// TwinCAT 3 PLC project Ciclo_di_Lavorazione
// ProgramVersion: 3.1.4023.0
// libraries:
//   Tc2_Standard, * (Beckhoff Automation GmbH)
//   Tc2_System, * (Beckhoff Automation GmbH)
//   Tc3_Module, * (Beckhoff Automation GmbH)
// project tree:
//   GVLs/ ZONE.TcGVL
//   / PlcTask.TcTTO
//   POUs/ MAIN.TcPOU, MASTER.TcPOU, Z2.TcPOU
// real-time tasks:
//   TASK PlcTask: cycle T#10ms, priority 20, ADS port 350

CONFIGURATION Ciclo_di_Lavorazione
    RESOURCE PLC ON TwinCAT3
        TASK PlcTask(INTERVAL := T#10ms, PRIORITY := 20);
        PROGRAM MAIN WITH PlcTask : MAIN;
    END_RESOURCE
END_CONFIGURATION

// ---- GVLs/ZONE.TcGVL
{attribute 'qualified_only'}
VAR_GLOBAL
db1 : BOOL;
Z2 : BOOL;
Db3 : BOOL;
Db4 : BOOL;
Db5 : BOOL;
Db6 : BOOL;
END_VAR

// ---- POUs/MAIN.TcPOU
PROGRAM MAIN
VAR
	START  : BOOL;
	STOP   : BOOL;
	EMERG  : BOOL := TRUE;
	ACK    : BOOL;
	MASTER : MASTER;
END_VAR

MASTER(START := IO.START, STOP := IO.STOP, EMERG := IO.EMERG, ACK := IO.ACK);
IO.H1 := MASTER.H1;
IO.H2 := MASTER.H2;
IO.H3 := MASTER.H3;

END_PROGRAM

// ---- POUs/MASTER.TcPOU
FUNCTION_BLOCK MASTER

VAR_INPUT
	START  : BOOL;
	STOP   : BOOL;
	EMERG  : BOOL;
	ACK    : BOOL;
END_VAR

VAR_OUTPUT
	H1         : BOOL;
	H2         : BOOL;
	H3     	   : BOOL;
	RIPRISTINO : BOOL;
END_VAR

VAR
END_VAR

VAR_STAT
	enable      : BOOL := FALSE;
	emergenza   : BOOL := FALSE;
	acknowledge : BOOL := FALSE;
END_VAR

IF(EMERG = FALSE) THEN
	enable := FALSE;
	emergenza := TRUE;
	H2 := TRUE;
	
ELSIF(emergenza = TRUE AND ACK = TRUE) THEN
	emergenza := FALSE;
	H2 := FALSE;
	H3 := TRUE;
	acknowledge := TRUE;
	
END_IF

IF(acknowledge = TRUE)
//	AND Db1.libero_O = TRUE
//	AND Z2.libero_O = TRUE
//	AND Db3.libero_O = TRUE
//	AND Db4.libero_O = TRUE
//	AND Db5.libero_O = TRUE
//	AND Db6.libero_O = TRUE)
 THEN
	
	acknowledge := FALSE;
	H3 := FALSE;
	H1 := FALSE;
END_IF

END_FUNCTION_BLOCK

// ---- POUs/Z2.TcPOU
FUNCTION_BLOCK Z2 
VAR_INPUT	
	ENABLE     : BOOL;
	EMG        : BOOL;
	RIPRISTINO : BOOL;
	LIBERO_I   : BOOL;
	TRIGGER_I  : BOOL;
a_0 : BOOL;
a_1	: BOOL;
I5 : BOOL;

END_VAR
VAR_OUTPUT
LIBERO_O   : BOOL;
TRIGGER_O  : BOOL;	
Q1 : BOOL;
Q2 : BOOL;

END_VAR

VAR	
stato : (S_attesa, S_uscita, S_Rientro, S_Ripristino, S_Emergenza) := S_attesa;
S_attesa : BOOL;
S_Uscita : BOOL;
S_rientro : BOOL;
S_ripristino : BOOL;
S_emergenza  : BOOL;
Trigger_OUT : TON();

END_VAR

//dichiarazione timer

Trigger_OUT(IN := Trigger_OUT.Q, PT := T#3S);

//Comandi transizione degli stati


IF EMG = FALSE  OR Enable = FALSE THEN
	
	stato := S_Emergenza;
	
END_IF

CASE stato OF
	S_Emergenza:
	
		IF Enable = TRUE AND Ripristino = TRUE THEN
		
			stato := S_Ripristino;
		
		END_IF
		
		Q1 := FALSE;
		Q2 := FALSE;
		Libero_O := FALSE;
		Trigger_O := FALSE;
	S_Ripristino:
		
		IF Enable = TRUE AND a_0 = TRUE THEN
			
			stato := S_Attesa;
			
		END_IF
		
		Q1 := TRUE;
		Q2 := FALSE;
		libero_O := FALSE;
		Trigger_O := FALSE;
	
	S_Attesa: 
	
		IF Enable = TRUE AND Trigger_I = TRUE AND Libero_I = TRUE AND a_0 = TRUE THEN
			
			stato := S_Uscita;
			
		END_IF
	
		Q1 := FALSE;
		Q2 := FALSE;
		Libero_O := TRUE;
		Trigger_O := FALSE;
	S_Uscita:
	
		IF a_1 = TRUE THEN
			
			stato := S_Rientro;
			
		END_IF
	
		Q1 := FALSE;
		Q2 := TRUE;
		Libero_O := FALSE;
		Trigger_O := FALSE;
	
S_Rientro:
	
		IF a_0 = TRUE THEN
			
			stato := S_Attesa;
			
		END_IF
	
		Q1 := TRUE;
		Q2 := FALSE;
		Libero_O := TRUE;
		Trigger_OUT.Q;
		Trigger_O := TRUE;
END_CASE

END_FUNCTION_BLOCK
